FUNCTION_BLOCK OutputChannelV2BOOL (* Basic Function Block Type *)
  (* Standard: 61499-2 *)
  (* Version 0.0, 12/03/2018, Atmojo, nxtControl GmbH, Template *)
  PACKAGE Main;
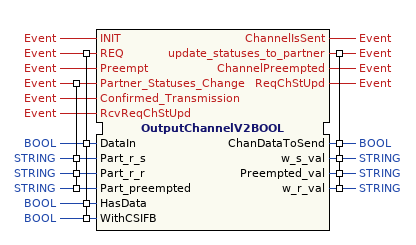
  EVENT_INPUT
    INIT;
    REQ WITH DataIn, HasData, WithCSIFB; (* Normal Execution Request *)
    Preempt;
    Partner_Statuses_Change WITH Part_r_s, Part_r_r, Part_preempted;
    Confirmed_Transmission;
    RcvReqChStUpd;
  END_EVENT
  EVENT_OUTPUT
    ChannelIsSent; (* Execution Confirmation *)
    update_statuses_to_partner WITH ChanDataToSend, w_s_val, Preempted_val, w_r_val;
    ChannelPreempted;
    ReqChStUpd;
  END_EVENT
  VAR_INPUT
    DataIn : BOOL;
    Part_r_s : STRING;
    Part_r_r : STRING;
    Part_preempted : STRING;
    HasData : BOOL;
    WithCSIFB : BOOL;
  END_VAR
  VAR_OUTPUT
    ChanDataToSend : BOOL;
    w_s_val : STRING := '0';
    Preempted_val : STRING := '0';
    w_r_val : STRING := '0';
  END_VAR
  VAR
    Part_r_s_localcopy : INT := 0;
    Part_r_r_localcopy : INT := 0;
    Part_preempted_localcopy : INT := 0;
    w_s : INT := 0;
    w_r : INT := 0;
    data_buffer : BOOL;
    Chan_Preempted_Status : INT := 0;
    Part_r_s_localcopy_other : INT;
    Part_r_r_localcopy_other : INT;
    Part_preempted_localcopy_other : INT;
    previous_w_s : INT;
    WaitingConfirmation : BOOL := FALSE;
    WithCSIFBStat : BOOL := FALSE;
  END_VAR
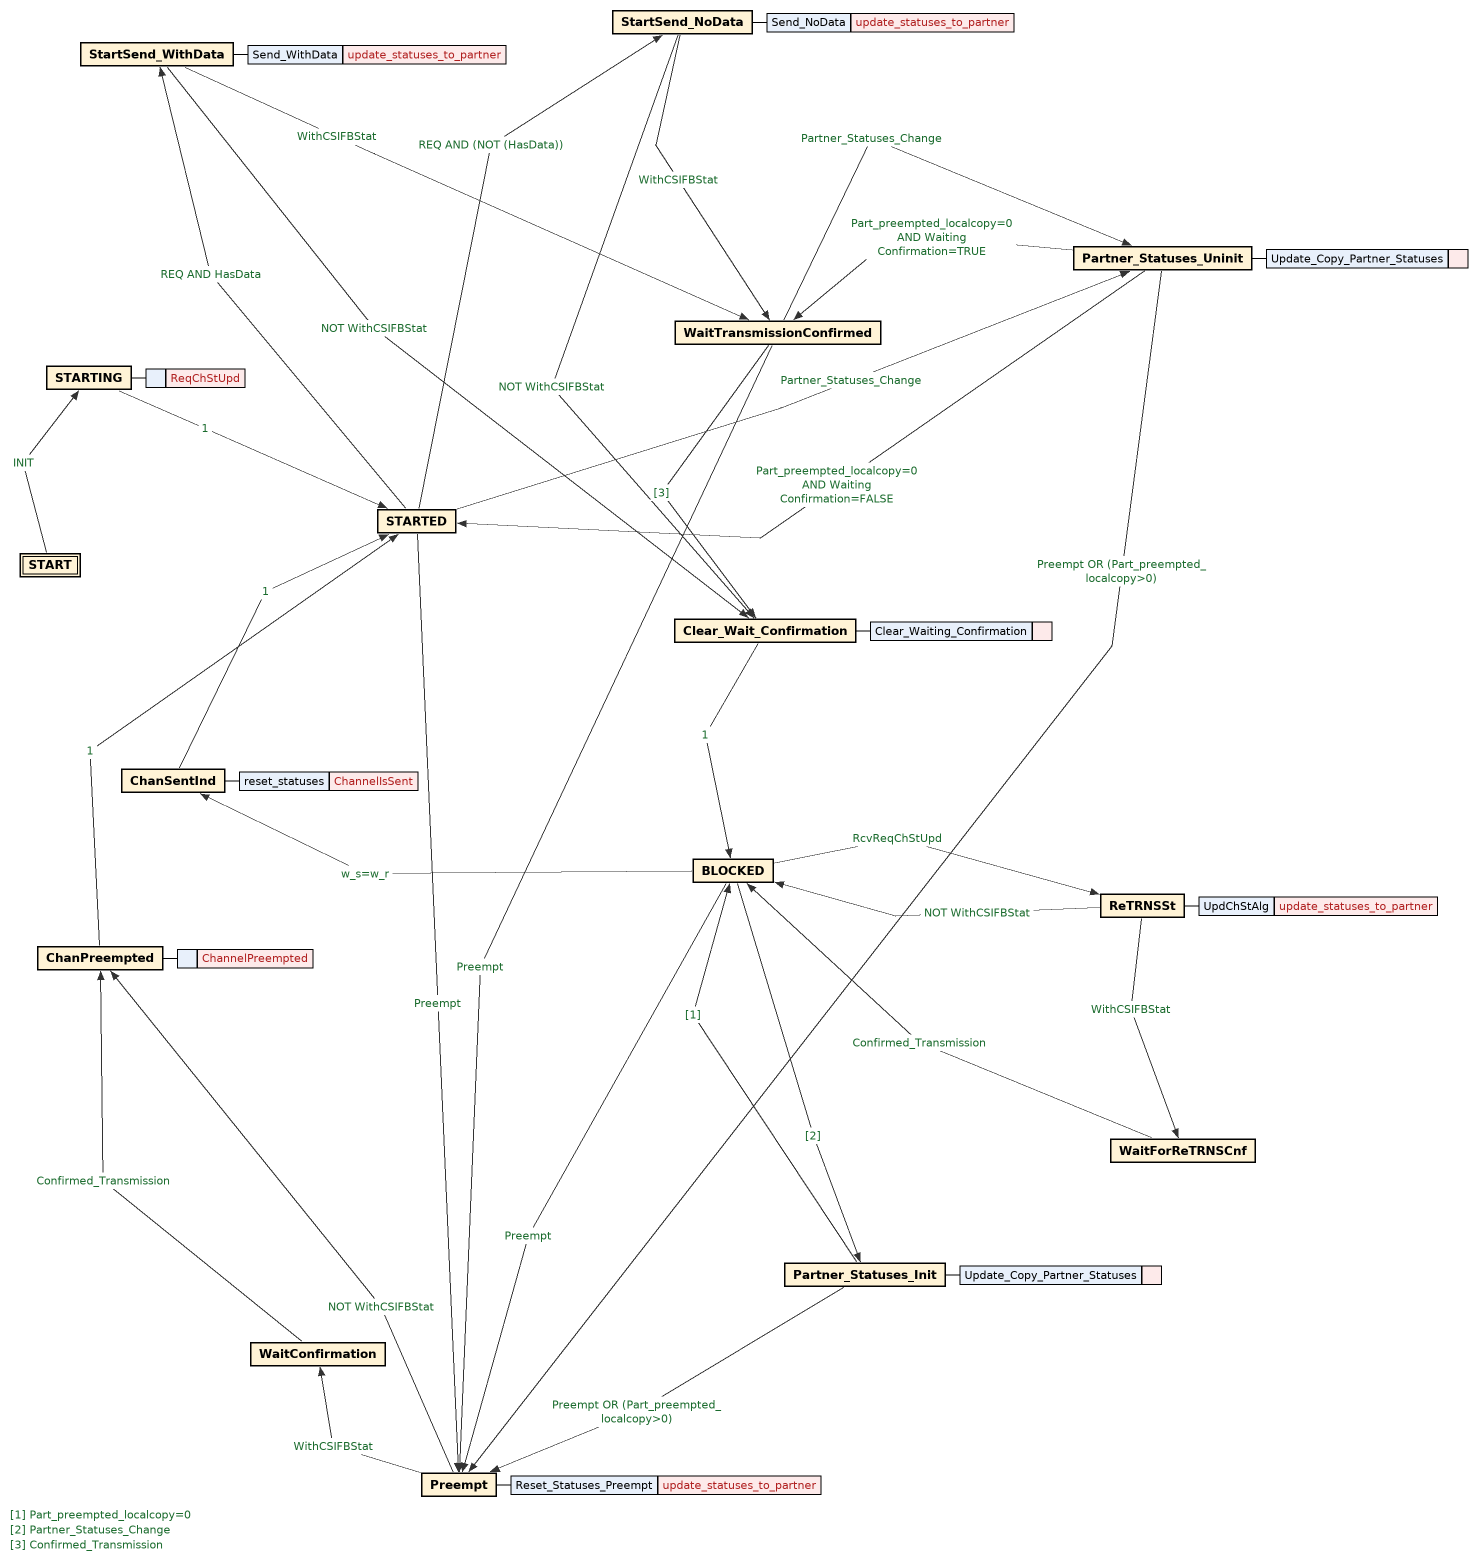
  EC_STATES
    START; (* Initial State *)
    StartSend_WithData : Send_WithData -> update_statuses_to_partner; (* Normal execution *)
    Preempt : Reset_Statuses_Preempt -> update_statuses_to_partner;
    BLOCKED;
    Partner_Statuses_Init : Update_Copy_Partner_Statuses;
    Partner_Statuses_Uninit : Update_Copy_Partner_Statuses;
    StartSend_NoData : Send_NoData -> update_statuses_to_partner;
    WaitTransmissionConfirmed;
    Clear_Wait_Confirmation : Clear_Waiting_Confirmation;
    ChanPreempted : -> ChannelPreempted;
    ChanSentInd : reset_statuses -> ChannelIsSent;
    WaitConfirmation;
    ReTRNSSt : UpdChStAlg -> update_statuses_to_partner;
    WaitForReTRNSCnf;
    STARTING : -> ReqChStUpd;
    STARTED;
  END_STATES
  EC_TRANSITIONS
    STARTED TO StartSend_WithData := REQ AND HasData;
    STARTED TO Preempt := Preempt;
    WaitConfirmation TO ChanPreempted := Confirmed_Transmission;
    BLOCKED TO Preempt := Preempt;
    BLOCKED TO Partner_Statuses_Init := Partner_Statuses_Change;
    Partner_Statuses_Init TO BLOCKED := Part_preempted_localcopy=0;
    Partner_Statuses_Init TO Preempt := Preempt OR (Part_preempted_localcopy>0);
    STARTED TO Partner_Statuses_Uninit := Partner_Statuses_Change;
    Partner_Statuses_Uninit TO STARTED := Part_preempted_localcopy=0 AND WaitingConfirmation=FALSE;
    Partner_Statuses_Uninit TO Preempt := Preempt OR (Part_preempted_localcopy>0);
    STARTED TO StartSend_NoData := REQ AND (NOT (HasData));
    WaitTransmissionConfirmed TO Clear_Wait_Confirmation := Confirmed_Transmission;
    StartSend_WithData TO WaitTransmissionConfirmed := WithCSIFBStat;
    StartSend_NoData TO WaitTransmissionConfirmed := WithCSIFBStat;
    WaitTransmissionConfirmed TO Partner_Statuses_Uninit := Partner_Statuses_Change;
    Partner_Statuses_Uninit TO WaitTransmissionConfirmed := Part_preempted_localcopy=0 AND WaitingConfirmation=TRUE;
    Clear_Wait_Confirmation TO BLOCKED := 1;
    ChanSentInd TO STARTED := 1;
    ChanPreempted TO STARTED := 1;
    WaitTransmissionConfirmed TO Preempt := Preempt;
    BLOCKED TO ChanSentInd := w_s=w_r;
    StartSend_WithData TO Clear_Wait_Confirmation := NOT WithCSIFBStat;
    StartSend_NoData TO Clear_Wait_Confirmation := NOT WithCSIFBStat;
    Preempt TO WaitConfirmation := WithCSIFBStat;
    Preempt TO ChanPreempted := NOT WithCSIFBStat;
    BLOCKED TO ReTRNSSt := RcvReqChStUpd;
    ReTRNSSt TO BLOCKED := NOT WithCSIFBStat;
    ReTRNSSt TO WaitForReTRNSCnf := WithCSIFBStat;
    WaitForReTRNSCnf TO BLOCKED := Confirmed_Transmission;
    START TO STARTING := INIT;
    STARTING TO STARTED := 1;
  END_TRANSITIONS
  ALGORITHM Send_WithData IN ST: (* Normally executed algorithm *)
  w_s:=w_s+1;
	previous_w_s:=w_s;
	data_buffer:=DataIn;
	w_s_val:= INT_TO_STRING(w_s);
	w_r_val:=INT_TO_STRING (w_r);
	Preempted_val:= INT_TO_STRING  (Chan_Preempted_Status);
	ChanDataToSend:=data_buffer;
	WaitingConfirmation:=TRUE;
	WithCSIFBStat:=WithCSIFB;
  END_ALGORITHM
  ALGORITHM Reset_Statuses_Preempt IN ST:
Preempted_val:= INT_TO_STRING (Chan_Preempted_Status+1);

w_s:=0;
w_r:=0;

Chan_Preempted_Status:=0;
Part_preempted_localcopy:=0;
WaitingConfirmation:=FALSE;

w_s_val:= INT_TO_STRING (w_s);
w_r_val:= INT_TO_STRING (w_r);
  END_ALGORITHM
  ALGORITHM Update_Copy_Partner_Statuses IN ST:
Part_r_r_localcopy:=STRING_TO_INT(Part_r_r);
Part_r_s_localcopy:=STRING_TO_INT(Part_r_s);
Part_preempted_localcopy:=STRING_TO_INT(Part_preempted);
w_r:=Part_r_s_localcopy;
w_s:=Part_r_r_localcopy;
  END_ALGORITHM
  ALGORITHM Update_Copy_Partner_Preempted_Status IN ST:
Part_preempted_localcopy:=STRING_TO_INT(Part_preempted);
  END_ALGORITHM
  ALGORITHM SendStatuses IN ST:
ChanDataToSend:=data_buffer;
w_s_val:=INT_TO_STRING(w_s);
w_r_val:=INT_TO_STRING(w_r);
Preempted_val:= INT_TO_STRING (Chan_Preempted_Status);
  END_ALGORITHM
  ALGORITHM Update_Copy_Partner_Statuses_Preempt IN ST:
Part_r_r_localcopy:=STRING_TO_INT(Part_r_r);
Part_r_s_localcopy:=STRING_TO_INT(Part_r_s);
Part_preempted_localcopy:=STRING_TO_INT(Part_preempted);
w_r:=Part_r_s_localcopy;
  END_ALGORITHM
  ALGORITHM reset_statuses IN ST:
w_s:=0;
w_r:=0;

Chan_Preempted_Status:=0;
Part_preempted_localcopy:=0;
WaitingConfirmation:=FALSE;
w_r_val:= '0';
w_s_val:='0';
Preempted_val:='0';
  END_ALGORITHM
  ALGORITHM Send_NoData IN ST:
previous_w_s:=w_s;
	w_s:=w_s+1;
	previous_w_s:=w_s;
	w_s_val:= INT_TO_STRING (w_s);
	w_r_val:= INT_TO_STRING (w_r);
	Preempted_val:=INT_TO_STRING (Chan_Preempted_Status);

	WaitingConfirmation:=TRUE;
	WithCSIFBStat:=WithCSIFB;
  END_ALGORITHM
  ALGORITHM Clear_Waiting_Confirmation IN ST:
WaitingConfirmation:=FALSE;
  END_ALGORITHM
  ALGORITHM UpdChStAlg IN ST:
w_s_val:= INT_TO_STRING(w_s);
	w_r_val:=INT_TO_STRING (w_r);
	Preempted_val:= INT_TO_STRING  (Chan_Preempted_Status);
	ChanDataToSend:=data_buffer;
  END_ALGORITHM
END_FUNCTION_BLOCK
